// TwinCAT 3 PLC project TC3_CNCPLCBase
// Title: CNC PLC Project
// Company: Beckhoff Automation GmbH & Co. KG
// Author: Beckhoff Automation GmbH & Co. KG
// ProjectVersion: 3.1.5000.18
// Description: TwinCAT CNC Base Project
// ProgramVersion: 3.1.4022.1
// libraries:
//   Tc2_CncHli, * (Beckhoff Automation GmbH)
//   Tc2_Standard, * (Beckhoff Automation GmbH)
//   Tc2_System, * (Beckhoff Automation GmbH)
//   Tc3_CNC, * (Beckhoff Automation GmbH)
//   Tc3_EventLogger, * (Beckhoff Automation GmbH)
//   Tc3_JsonXml, * (Beckhoff Automation GmbH)
//   Tc3_Module, * (Beckhoff Automation GmbH)
// project tree:
//   CNC/ Global_CNC.TcGVL, PRG_CNCAxesHandler.TcPOU, PRG_CNCChannelHandler.TcPOU, PRG_CNCManualMode.TcPOU, PRG_CNCVariablesViewer.TcPOU, PRG_ManualFnc.TcPOU
//   / FAST.TcPOU, MAIN.TcPOU, PlcFastTask.TcTTO, PlcTask.TcTTO
//   HMI/ Global_HMI.TcGVL, ST_MachineData.TcDUT, ST_MachineMode.TcDUT, ST_MANUAL.TcDUT, ST_Position.TcDUT
//   Messages/ FB_Alarm.TcPOU, FB_ExtSimpleEventLog.TcPOU, FB_SimpleEventLog.TcPOU, Global_Messages.TcGVL, PRG_Messages.TcPOU, PRG_MessagesV2.TcPOU
//   Samples/ PRG_FastMFunctions.TcPOU
// real-time tasks:
//   TASK PlcTask: cycle T#10ms, priority 20, ADS port 350
//   TASK PlcFastTask: cycle T#10ms, priority 21, ADS port 351
// motion (NC):
//   TASK NC-Task 1 SAF: cycle T#2ms, priority 4, ADS port 501
//   TASK NC-Task 1 SVB: cycle T#10ms, priority 9, ADS port 511
//   AXIS RollerVibrator (id 1)
//     General: UnitName=Degree
//     Dynamic: AccelerationMaximum=72000, DecelerationMaximum=72000, Acceleration=72000, Deceleration=72000, Jerk=432000
//     Velo: RefSearch=313.26, RefSync=313.26, SlowManual=1566.3, FastManual=9397.8, Fast=31326, Maximum=60000
//     PositionAreaControl: Range=10
//     OtherSettings: AllowMotionCmdToSlave=true, PulseDistancePos=10, PulseDistanceNeg=10
//     encoder EncType=19
//       EncPara: ScaleFactorNumerator=360, ScaleFactorDenominator=1048576, MaxCount=#xffffffff
//     drive DrvType=16
//       DrvPara: MaxCount=#xffffffff, DriveControlDWord=#x00020000
//         Analog: VeloReferenz=36000, VeloScale=32, TorqueSetpointScale=10, ScaleFactorActTorque=0.1
//         TimeComp: TaskDelayCycles=1
//     controller CtrType=1
//       CtrPara: PriorControlFactor=1
//         PosDiffControl: Enable=false, Range=10
//         Observer: BandWidth=20
//   AXIS RollerCompactor (id 2)
//     General: UnitName=Degree
//     Dynamic: AccelerationMaximum=72000, DecelerationMaximum=72000, Acceleration=72000, Deceleration=72000, Jerk=432000
//     Velo: RefSearch=313.26, RefSync=313.26, SlowManual=1566.3, FastManual=9397.8, Fast=31326, Maximum=60000
//     PositionAreaControl: Range=10
//     OtherSettings: AllowMotionCmdToSlave=true, PulseDistancePos=10, PulseDistanceNeg=10
//     encoder EncType=19
//       EncPara: ScaleFactorNumerator=360, ScaleFactorDenominator=1048576, MaxCount=#xffffffff
//     drive DrvType=16
//       DrvPara: MaxCount=#xffffffff, DriveControlDWord=#x00020000
//         Analog: VeloReferenz=36000, VeloScale=32, TorqueSetpointScale=10, ScaleFactorActTorque=0.1
//         TimeComp: TaskDelayCycles=1
//     controller CtrType=1
//       CtrPara: PriorControlFactor=1
//         PosDiffControl: Enable=false, Range=10
//         Observer: BandWidth=20
// I/O:
//   DEVICE Device 1 (EtherCAT), AmsNetId 5.85.147.42.2.1
//     Term 1 (EK1200) [EK1200-5000 EtherCAT Power supply (2A E-Bus)]
//       Term 2 (EK1122) [EK1122 2 port EtherCAT junction]
//         Term 3 (EK1100) [EK1100 EtherCAT Coupler (2A E-Bus)]
//         Drive 4 (ctrlX DRIVE XCD (SoE) 1/2) [ctrlX DRIVE XCD (SoE) Axis 1 of 2]
//         Drive 5 (ctrlX DRIVE XCD (SoE) 2/2) [ctrlX DRIVE XCD (SoE) Axis 2 of 2]
//         Drive 6 (ctrlX DRIVE XMD (SoE) 1/2) [ctrlX DRIVE XMD (SoE) Axis 1 of 2]
//         Drive 7 (ctrlX DRIVE XMD (SoE) 2/2) [ctrlX DRIVE XMD (SoE) 2 of 2]
//         Drive 8 (ctrlX DRIVE XMD (SoE) 1/2) [ctrlX DRIVE XMD (SoE) Axis 1 of 2]
//         Drive 9 (ctrlX DRIVE XMD (SoE) 2/2) [ctrlX DRIVE XMD (SoE) 2 of 2]
//         Drive 10 (ctrlX DRIVE XMS (SoE)) [ctrlX DRIVE XMS (SoE)]
//         Drive 24 (IndraDrive MPB20 FSoE) [IndraDrive MPB20 FSoE]
//         Term 26 (EK1100) [EK1100 EtherCAT Coupler (2A E-Bus)]
//           Term 27 (EL4124) [EL4124 4Ch. Ana. Output 4-20mA, 16bit]
//           Term 28 (EL2008) [EL2008 8Ch. Dig. Output 24V, 0.5A]
//           Term 32 (EL9011) [EL9011 End Terminal]
//       Term 29 (EK1122) [EK1122 2 port EtherCAT junction]
//         Term 30 (EK1100) [EK1100 EtherCAT Coupler (2A E-Bus)]
//           Term 31 (EL7211-9014) [EL7211-9014 1Ch. MDP742 Servo motor output stage with OCT (50V, 4.5A RMS) and STO input]
//           Term 32 (EL7211-9014) [EL7211-9014 1Ch. MDP742 Servo motor output stage with OCT (50V, 4.5A RMS) and STO input]
//           Term 33 (EL9011) [EL9011 End Terminal]
//   DEVICE Device 4 (RT-Ethernet Protocol), AmsNetId 5.85.147.42.5.1
//   DEVICE Device 3 (USB)
//     Box 1 (CX2100 Power Supply)
//   DEVICE Device 5 (NOV-DP-RAM)
// variable links:
//   CNC/Axes/A <-> Device 1 (EtherCAT)/Term 1 (EK1200)/Term 2 (EK1122)/Drive 24 (IndraDrive MPB20 FSoE)
//     Inputs/Drive status word <-> AT/Drive status word
//     Inputs/Position feedback value 1 <-> AT/Position feedback value 1
//     Inputs/WcState <-> WcState/WcState
//     Outputs/Master control word <-> MDT/Master control word
//     Outputs/Position command value <-> MDT/Position command value
//   CNC/Axes/X0_M <-> Device 1 (EtherCAT)/Term 1 (EK1200)/Term 2 (EK1122)/Drive 4 (ctrlX DRIVE XCD (SoE) 1/2)
//     Inputs/Drive status word <-> AT/Drive status word
//     Inputs/Position feedback value 1 <-> AT/Position feedback value 1
//     Inputs/Power supply status word <-> AT/Power supply status word
//     Inputs/WcState <-> WcState/WcState
//     Outputs/Master control word <-> MDT/Master control word
//     Outputs/Position command value <-> MDT/Position command value
//     Outputs/Power supply control word <-> MDT/Power supply control word
//   CNC/Axes/X0_S <-> Device 1 (EtherCAT)/Term 1 (EK1200)/Term 2 (EK1122)/Drive 5 (ctrlX DRIVE XCD (SoE) 2/2)
//     Inputs/Drive status word <-> AT/Drive status word
//     Inputs/Position feedback value 1 <-> AT/Position feedback value 1
//     Inputs/WcState <-> WcState/WcState
//     Outputs/Master control word <-> MDT/Master control word
//     Outputs/Position command value <-> MDT/Position command value
//   CNC/Axes/X1_M <-> Device 1 (EtherCAT)/Term 1 (EK1200)/Term 2 (EK1122)/Drive 6 (ctrlX DRIVE XMD (SoE) 1/2)
//     Inputs/Device control: Status word <-> AT/Device control: Status word
//     Inputs/Drive status word <-> AT/Drive status word
//     Inputs/Position feedback value 1 <-> AT/Position feedback value 1
//     Inputs/WcState <-> WcState/WcState
//     Outputs/DC Bus Power Control <-> MDT/DC Bus Power Control
//     Outputs/Master control word <-> MDT/Master control word
//     Outputs/Position command value <-> MDT/Position command value
//   CNC/Axes/X1_S <-> Device 1 (EtherCAT)/Term 1 (EK1200)/Term 2 (EK1122)/Drive 7 (ctrlX DRIVE XMD (SoE) 2/2)
//     Inputs/Device control: Status word <-> AT/Device control: Status word
//     Inputs/Drive status word <-> AT/Drive status word
//     Inputs/Position feedback value 1 <-> AT/Position feedback value 1
//     Inputs/WcState <-> WcState/WcState
//     Outputs/DC Bus Power Control <-> MDT/DC Bus Power Control
//     Outputs/Master control word <-> MDT/Master control word
//     Outputs/Position command value <-> MDT/Position command value
//   CNC/Axes/Y <-> Device 1 (EtherCAT)/Term 1 (EK1200)/Term 2 (EK1122)/Drive 10 (ctrlX DRIVE XMS (SoE))
//     Inputs/Device control: Status word <-> AT/Device control: Status word
//     Inputs/Drive status word <-> AT/Drive status word
//     Inputs/Position feedback value 1 <-> AT/Position feedback value 1
//     Inputs/WcState <-> WcState/WcState
//     Outputs/DC Bus Power Control <-> MDT/DC Bus Power Control
//     Outputs/Master control word <-> MDT/Master control word
//     Outputs/Position command value <-> MDT/Position command value
//   CNC/Axes/Z_M <-> Device 1 (EtherCAT)/Term 1 (EK1200)/Term 2 (EK1122)/Drive 8 (ctrlX DRIVE XMD (SoE) 1/2)
//     Inputs/Device control: Status word <-> AT/Device control: Status word
//     Inputs/Drive status word <-> AT/Drive status word
//     Inputs/Position feedback value 1 <-> AT/Position feedback value 1
//     Inputs/WcState <-> WcState/WcState
//     Outputs/DC Bus Power Control <-> MDT/DC Bus Power Control
//     Outputs/Master control word <-> MDT/Master control word
//     Outputs/Position command value <-> MDT/Position command value
//   CNC/Axes/Z_S <-> Device 1 (EtherCAT)/Term 1 (EK1200)/Term 2 (EK1122)/Drive 9 (ctrlX DRIVE XMD (SoE) 2/2)
//     Inputs/Device control: Status word <-> AT/Device control: Status word
//     Inputs/Drive status word <-> AT/Drive status word
//     Inputs/Position feedback value 1 <-> AT/Position feedback value 1
//     Inputs/WcState <-> WcState/WcState
//     Outputs/DC Bus Power Control <-> MDT/DC Bus Power Control
//     Outputs/Master control word <-> MDT/Master control word
//     Outputs/Position command value <-> MDT/Position command value
//   NC-Task 1 SAF/Axes/RollerCompactor <-> Device 1 (EtherCAT)/Term 1 (EK1200)/Term 29 (EK1122)/Term 30 (EK1100)/Term 32 (EL7211-9014)
//     Drive/Inputs/In/nDcOutputTime <-> InfoData/DcOutputShift
//     Drive/Inputs/In/nState1 <-> DRV Statusword/Statusword
//     Drive/Inputs/In/nState2 <-> DRV Statusword/Statusword @bit 8
//     Drive/Inputs/In/nState4 @bit 1 <-> WcState/InputToggle
//     Drive/Inputs/In/nState4 <-> WcState/WcState
//     Drive/Outputs/Out/nCtrl1 <-> DRV Controlword/Controlword
//     Drive/Outputs/Out/nCtrl2 <-> DRV Controlword/Controlword @bit 8
//     Drive/Outputs/Out/nDataOut2 <-> DRV Target velocity/Target velocity
//     Enc/Inputs/In/nDataIn1 <-> FB Position/Position
//     Enc/Inputs/In/nDcInputTime <-> InfoData/DcInputShift
//     Enc/Inputs/In/nState4 @bit 1 <-> WcState/InputToggle
//     Enc/Inputs/In/nState4 <-> WcState/WcState
//   NC-Task 1 SAF/Axes/RollerVibrator <-> Device 1 (EtherCAT)/Term 1 (EK1200)/Term 29 (EK1122)/Term 30 (EK1100)/Term 31 (EL7211-9014)
//     Drive/Inputs/In/nDcOutputTime <-> InfoData/DcOutputShift
//     Drive/Inputs/In/nState1 <-> DRV Statusword/Statusword
//     Drive/Inputs/In/nState2 <-> DRV Statusword/Statusword @bit 8
//     Drive/Inputs/In/nState4 @bit 1 <-> WcState/InputToggle
//     Drive/Inputs/In/nState4 <-> WcState/WcState
//     Drive/Outputs/Out/nCtrl1 <-> DRV Controlword/Controlword
//     Drive/Outputs/Out/nCtrl2 <-> DRV Controlword/Controlword @bit 8
//     Drive/Outputs/Out/nDataOut2 <-> DRV Target velocity/Target velocity
//     Enc/Inputs/In/nDataIn1 <-> FB Position/Position
//     Enc/Inputs/In/nDcInputTime <-> InfoData/DcInputShift
//     Enc/Inputs/In/nState4 @bit 1 <-> WcState/InputToggle
//     Enc/Inputs/In/nState4 <-> WcState/WcState

CONFIGURATION TC3_CNCPLCBase
    RESOURCE PLC ON TwinCAT3
        TASK PlcFastTask(INTERVAL := T#10ms, PRIORITY := 21);
        TASK PlcTask(INTERVAL := T#10ms, PRIORITY := 20);
        PROGRAM FAST WITH PlcFastTask : FAST;
        PROGRAM MAIN WITH PlcTask : MAIN;
    END_RESOURCE
END_CONFIGURATION

// ---- HMI/ST_MachineData.TcDUT
TYPE ST_MachineData :
STRUCT
	// @1: Value1
	Value1: INT;
	// @1: Bool Value
	Value2: bool;
	// @1: Position
	pos : ST_Position;
	// @1: Manual @6:1
	manualFunction : ST_Manual;
END_STRUCT
END_TYPE

// ---- HMI/ST_MachineMode.TcDUT
TYPE ST_MachineMode :
STRUCT
	/// Operation Mode 
	Standby: BOOL;
	Manual: BOOL;
	MDI: BOOL;
	Automatic: BOOL;
	///REFERENCE		: BOOL;  TC3HR
	Homing: BOOL;
	/// Operation State
	Select : BOOL; 
	Ready  : BOOL;
	Start: BOOL;
	Stop: BOOL;
	Reset: BOOL;
	Error: BOOL;
	/// Special functions 
	ChannelSignals: ST_ChannelSignals;
	BlockSearch: ST_BlockSearch;
	SyntaxCheck: ST_SyntaxCheck;
	ManualMode: ST_ManualMode;
	/// Strings 
//	ProgramName: STRING(1024);
//	MDIString: STRING(1024);
	ProgramName: STRING(HLI_IMCM_MODE_STATE_PARAM_STRL);
	MDIString: STRING(HLI_IMCM_MODE_STATE_PARAM_STRL);

END_STRUCT
END_TYPE

// ---- HMI/ST_MANUAL.TcDUT
TYPE ST_MANUAL :
STRUCT
	// @1:cylinder one @2:on:1 @3:off:1 @4:pos1:1 @5:pos2:0
	cyl1 			: BYTE;	
	cyl1Status		: BYTE;
	
	// @1:conveyor @2:IMG1:1 @2:IMG2 @3:IMG15 @4:IMG16 @5:IMG7 @6:IMG13 @7:IMG14
	conv 			: BYTE;
	convStatus 		: BYTE;
	
	
END_STRUCT
END_TYPE

// ---- HMI/ST_Position.TcDUT
TYPE ST_Position :
STRUCT
	// @1:X
	x	:	LREAL;
	// @1:Y
	y	: 	LREAL;
	// @1:Z	
	Z	: 	LREAL;
END_STRUCT
END_TYPE

// ---- CNC/Global_CNC.TcGVL
VAR_GLOBAL CONSTANT
	// Max index of channel that is used starting at 0, example: 1 -> totally 2 channels, maximum of 11 (12 channels) is allowed here
	MAX_USED_CHANNEL_IDX		: INT := 2;									
	libVersion					: ST_LibVersion := stLibVersion_Tc3_CNC;  	 
END_VAR

// ---- HMI/Global_HMI.TcGVL
VAR_GLOBAL
	/// HMI -> PLC 
	PLCChannelSignals: ST_ChannelSignals;
	/// HMI -> PLC 
	PLCSelectedChannel: INT := 0;
	/// HMI -> PLC 
	PLCFeedOverride: UINT := 100;
	/// HMI -> PLC 
	PLCSpindleOverride: UINT := 100;
	/// HMI -> PLC 
	PLCAxisEnable: BOOL;
	/// PLC -> HMI  
	PLCStatusAxisEnabled : BOOL;	
	/// HMI -> PLC 
	PLCReset: BOOL;
	PLCMachineMode: ARRAY[0..MAX_USED_CHANNEL_IDX] OF ST_MachineMode;
	/// PLC -> HMI : angewähltes File 
	PLCToHmiFile: STRING(255);
	/// Variablen für das Module "InformPlc" 
	bToggle: BOOL;
	sActualForm: STRING(255);
	nUserLevel: INT;
	sUserName: STRING(255);
	/// steigende Flanke: Applikation beenden 
	bExitApp: BOOL;	
	
	userActivity : BOOL;
	
	// @1:MachineData
	MachineData : ST_MachineData;
	
	// spindle manual mode
	nSpindleRpm:	DINT;	
	bSpindleStart: BOOL;
	bSpindleStop: BOOL;
	
	ManualFnc : ARRAY[0..3] OF FB_ManualFncFull;
	
END_VAR

// ---- Messages/Global_Messages.TcGVL
VAR_GLOBAL
	///--------------------------
	///	Messages                
	///--------------------------
	MSG_WARNING_List: ARRAY[FIRST_MESSAGE..LAST_MESSAGE] OF BOOL;
	MSG_WARNING_ListQuit: ARRAY[FIRST_MESSAGE..LAST_MESSAGE] OF BOOL;	
	MSG_ALARM_List: ARRAY[FIRST_MESSAGE..LAST_MESSAGE] OF BOOL;
	MSG_ALARM_ListQuit: ARRAY[FIRST_MESSAGE..LAST_MESSAGE] OF BOOL;			
END_VAR

VAR_GLOBAL CONSTANT
	FIRST_MESSAGE: UDINT := 1;
	LAST_MESSAGE: UDINT := 50;	
END_VAR

// ---- FAST.TcPOU
PROGRAM FAST
VAR
	nChan : INT;
	MOS_TS: INT;
	i: INT;	
	ChannelMHTFunction : ARRAY[0..MAX_USED_CHANNEL_IDX] OF HLI3_QuitChannelMHTFunction;
END_VAR

(****************************************************************************************)
(*	  							Wait for HLI initialization								*)
(****************************************************************************************)
IF NOT CNCSystem.bHLIInit THEN
	RETURN;
END_IF

IF PRG_CNCChannelHandler.stOptions.bDisableMFunctHandling THEN
	FOR i := 0 TO MAX_USED_CHANNEL_IDX DO
		ChannelMHTFunction[i](nChanIdx:=0, bM30Acknowledgement := TRUE);
	END_FOR
END_IF	

(* Programm call for MOS_TS M functions *)
// PRG_FastMFunctions();

END_PROGRAM

// ---- CNC/PRG_CNCChannelHandler.TcPOU
PROGRAM PRG_CNCChannelHandler
VAR	
	nChan					: INT;
	nOldSelectedChannel		: UDINT;
	CNCChannel				: ARRAY[0..MAX_USED_CHANNEL_IDX] OF HLI3_CNCChannel;	
	BlockSearch_Channel		: ARRAY[0..MAX_USED_CHANNEL_IDX] OF HLI3_BlockSearch;
	ErrorHandler_Channel	: ARRAY[0..MAX_USED_CHANNEL_IDX] OF FB_ChannelError;
	nChanNo: UDINT;	
	i: INT;	
	stOptions				: ST_CNC_CH_Options;
END_VAR

(****************************************************************************************)
(* POU:		PRG_ChannelHandler                     										*)
(* Type:	PRG																			*)
(* Author: 	HR / TV / MiB                                          						*)
(* Date: 	23.01.11																	*)
(* Last:	29.03.18																	*)
(* Rev.: 	1.6                                              							*)
(* ------------------------------------------------------------------------------------ *)
(* Desc:	Description																	*)
(****************************************************************************************)

(****************************************************************************************)
(*	  Map CNC function selection from HMI to selected channel (and state vice versa)  	*)
(****************************************************************************************)
IF (nOldSelectedChannel <>INT_TO_UDINT(PLCSelectedChannel)) THEN
	PLCChannelSignals.SingleBlock 		:= PLCMachineMode[PLCSelectedChannel].ChannelSignals.SingleBlock;
	PLCChannelSignals.PrgBlockIgnore	:= PLCMachineMode[PLCSelectedChannel].ChannelSignals.PrgBlockIgnore;
	PLCChannelSignals.M01Stop 			:= PLCMachineMode[PLCSelectedChannel].ChannelSignals.M01Stop;
	PLCChannelSignals.Backward 			:= PLCMachineMode[PLCSelectedChannel].ChannelSignals.Backward;
	PLCChannelSignals.FeedHold 			:= PLCMachineMode[PLCSelectedChannel].ChannelSignals.FeedHold;
	nOldSelectedChannel 				:= INT_TO_UDINT(PLCSelectedChannel);
END_IF

PLCMachineMode[PLCSelectedChannel].ChannelSignals.SingleBlock 		:= PLCChannelSignals.SingleBlock;
PLCMachineMode[PLCSelectedChannel].ChannelSignals.PrgBlockIgnore 	:= PLCChannelSignals.PrgBlockIgnore;
PLCMachineMode[PLCSelectedChannel].ChannelSignals.M01Stop 			:= PLCChannelSignals.M01Stop;
PLCMachineMode[PLCSelectedChannel].ChannelSignals.Backward 		:= PLCChannelSignals.Backward;
PLCMachineMode[PLCSelectedChannel].ChannelSignals.FeedHold 		:= PLCChannelSignals.FeedHold;


stOptions.bReferenceModeStartRequired := FALSE;

FOR i := 0 TO MAX_USED_CHANNEL_IDX DO
		
	nChan := i;	
	IF (HLI3_CheckChannelValid(nChan)) THEN		
		
		(* Error handler for channel 1 *)
		ErrorHandler_Channel[nChan](nChanIdx			:= nCHan);				
				
		(* Channel interface *)
		CNCChannel[nChan]
			(nChanIdx			:= nChan,							
			 // Operation Mode with VAR_IN_OUT Variables 
			 bModeStandby		:= PLCMachineMode[nChan].Standby,
			 bModeAutomatic		:= PLCMachineMode[nChan].Automatic,
			 bModeManual		:= PLCMachineMode[nChan].Manual,
			 bModeMDI			:= PLCMachineMode[nChan].MDI,	 
			 bModeReference		:= PLCMachineMode[nChan].Homing,
			 // Operation State with VAR_IN_OUT Variables
			 bStateSelect		:= PLCMachineMode[nChan].Select,
			 bStateReady		:= PLCMachineMode[nChan].Ready,
			 bStateStart		:= PLCMachineMode[nChan].Start,
			 bStateStop			:= PLCMachineMode[nChan].Stop,
			 bStateReset		:= PLCMachineMode[nChan].Reset,
			 // Operation Mode with VAR_IN Varaibles, the command is executed with a rising edge 
			 bCmdAutomatic 		:= FALSE,
			 bCmdManual 		:= FALSE,
    		 bCmdReference 		:= FALSE,
    		 bCmdMDI 			:= FALSE,		
			 // Operation State with VAR_IN Varaibles, the command is executed with a rising edge
			 bCmdStart 			:= FALSE,
			 bCmdStop  			:= FALSE,
	         bCmdReset 			:= FALSE,					 			 
			 // EmergencyStop 
			 bEmergencyStop 	:= FALSE,		(* If TRUE the interpolation will be aborted, Signal is no TwinSAFE function !*)
			 // Override 
			 nFeedOverride		:= PLCFeedOverride * 10,
			 nRapidFeedOverride := PLCFeedOverride * 10, 
			 // Special Functions 
			 sProgramName		:= PLCMachineMode[nChan].ProgramName,			 
			 sMDIString			:= PLCMachineMode[nChan].MDIString,
			 bBackwardMotion	:= PLCMachineMode[nChan].ChannelSignals.Backward,
			 bPrgBlockIgnore	:= PLCMachineMode[nChan].ChannelSignals.PrgBlockIgnore,
			 bFeedHold			:= PLCMachineMode[nChan].ChannelSignals.FeedHold,
			 bSingleBlock		:= PLCMachineMode[nChan].ChannelSignals.SingleBlock,
			 bDoSingleBlock		:= PLCMachineMode[nChan].ChannelSignals.DoSingleBlock,
			 bM01Stop			:= PLCMachineMode[nChan].ChannelSignals.M01Stop,
			 nSyntaxCheck		:= PLCMachineMode[nChan].SyntaxCheck.nType,
			 bM30Acknowledgement:= TRUE,
			 // Manual Mode 			 						 
			 stManualModeParameter  	 	 := stManualModeParameter[nChan],
			 stManualModeControlElements	 := stManualModeControlElements[nChan],
			 stManualModeControlElementState := stManualModeControlElementState,
			 // Options
			 stOptions			:= 	stOptions			 			 
			);
		
		(* Handle block search *)
		BlockSearch_Channel[nChan]
			(nChanIdx			:= nChan,
			 bStartRead      	:= PLCMachineMode[nChan].BlockSearch.bStartRead,   (* Edge signal *)
			 bStartWrite     	:= PLCMachineMode[nChan].BlockSearch.bStartWrite,  (* Edge signal *)
			 BlockSearch		:= PLCMachineMode[nChan].BlockSearch
			);
		
		CNCSystem.Channel[nChan].ActDistance 	:= DINT_TO_LREAL(BlockSearch_Channel[nChan].coveredDistance_AfterReset) / 10.0;
		CNCSystem.Channel[nChan].ActBlockCount 	:= BlockSearch_Channel[nChan].actualBlockCount_AfterReset;
						
	END_IF
END_FOR

END_PROGRAM

// ---- MAIN.TcPOU
PROGRAM MAIN
VAR
  
END_VAR

HLI3_Init(); 
PRG_Messages();  	// Messages Eventlogger V1
PRG_MessagesV2();   // Messages Eventlogger V2

(* Call CNC related code only if the HLI has been initialized succesfully! *)
IF CNCSystem.bHLIInit THEN
	PRG_CNCAxesHandler();    	
	PRG_CNCManualMode();
	PRG_CNCChannelHandler();	
	PRG_CNCVariablesViewer();
	PRG_ManualFnc();		
END_IF
(* Reset the reset flag from HMI *)
PLCReset := FALSE;

END_PROGRAM

// ---- Messages/PRG_Messages.TcPOU
PROGRAM PRG_Messages
VAR
	bStart: BOOL;
	fbWarningMessages : FB_SimpleEventLog;
	fbAlarmMessages : FB_SimpleEventLog;
	//fbExAlarmMessages : FB_ExtSimpleEventLog;
END_VAR

(*
	TCEVENTCLASS_NONE			:=0,	 No class
	TCEVENTCLASS_MAINTENANCE	:=1,	 Maintenance hint
	TCEVENTCLASS_MESSAGE		:=2,	 Message
	TCEVENTCLASS_HINT			:=3,	 Hint
	TCEVENTCLASS_STATEINFO		:=4,	 State information
	TCEVENTCLASS_INSTRUCTION	:=5,	 Instruction
	TCEVENTCLASS_WARNING		:=6,	 Warning
	TCEVENTCLASS_ALARM			:=7,	 Alarm
	TCEVENTCLASS_PARAMERROR		:=8	 Parameter error
*)


(* Shows how to generate messages *)
IF NOT bStart THEN
	bStart 				:= TRUE;

	fbWarningMessages
		(Init			:= TRUE,
		 SourceId		:= 51,
		 Class			:= TCEVENTCLASS_WARNING,
		 QuitRequireD	:= FALSE,
		 adrAlarmArray	:= ADR(MSG_WARNING_List),
		 adrQuitArray	:= ADR(MSG_WARNING_ListQuit)
		);

	fbAlarmMessages
		(Init			:= TRUE,
		 SourceId		:= 50,
		 Class			:= TCEVENTCLASS_ALARM,
		 QuitRequired	:= FALSE,
		 adrAlarmArray 	:= ADR(MSG_ALARM_List),
		 adrQuitArray	:= ADR(MSG_ALARM_ListQuit)
		);
		(*
		fbExAlarmMessages(
			Init:= TRUE, 
			SourceId:= 52,
			Class:= TCEVENTCLASS_WARNING, 				
			QuitRequired:= FALSE, 
			adrAlarmArray:= ADR(MSG_ExALARM_List), 
			adrQuitArray:= ADR(MSG_ExALARM_ListQuit), 
			adrEventData:= ADR(MSG_ExALARM_EventData),	 
			sFormatString:= '%d%s'		  
			);
			*)
ELSE
	fbWarningMessages
		(Init			:= FALSE);

	fbAlarmMessages
		(Init			:= FALSE);	
		(*
	fbExAlarmMessages
		(Init			:= FALSE);
*)	
END_IF

END_PROGRAM

// ---- Messages/FB_SimpleEventLog.TcPOU
///****************************************************************************************
///Name:				FB_SimpleEventLog
///Date:				13.10.2004
///Author:			Dirk Nordberg (BECKHOFF INDUSTRIE ELEKTRONIK)
///
///Description: Function block to control the EventLogger
///	Messages can be activated or deactivated through an array of bool.
///	The subscription of the array is equivalent to EventID from EventLogger.
///	Function block will be initialized with Init flag, then the busy flag is set true. 
///
///	Revision:	1.4
///	History:		13.10.2004	Ng	start coding
///					17.04.2005	MK	runtime optimized
///					07.07.2005	MK	short puls BF
///				    29.11.2010 	MiB  quittierungspflichtige Merker funktionieren nun wieder
///                 21.06.2013  TV   change : data type for pointer address from uint to pointer of int 
///****************************************************************************************
FUNCTION_BLOCK FB_SimpleEventLog
VAR_INPUT
	/// Rising flag starts the initialization 
	Init: BOOL;
	/// Number of the source Id 
	SourceId: UINT;
	/// Alarm error class 
	Class: UINT;
	/// Activate or deaktivate confirmation 
	QuitRequired: BOOL;
	/// Adress of the array for the messages 
	adrAlarmArray: POINTER TO BOOL;
	/// ...with constant boundaries ARRAY_LBOUND to ARRAY_UBOUND for array size 
	adrQuitArray: POINTER TO BOOL;
END_VAR
VAR_OUTPUT
	Busy: BOOL;
	Err: BOOL;
	ErrId: UDINT;
END_VAR
VAR CONSTANT
	ARRAY_LBOUND: UDINT := FIRST_MESSAGE;
	ARRAY_UBOUND: UDINT := LAST_MESSAGE;
	TCEVENTDATAFORMATSTRING: STRING := ' ';
	STATE_INIT: INT := 0;
	STATE_IDLE: INT := 1;
	STATE_RESET_EVENT: INT := 2;
	STATE_QUIT_EVENT: INT := 3;
	STATE_RESET_END: INT := 4;
	STATE_WAIT: INT := 5;
END_VAR
VAR
	state: INT;
	///{flag nowatch on }
	bReady: BOOL := TRUE;
	nMsgHasChanged: DINT;
	bEvtState: ARRAY[ARRAY_LBOUND..ARRAY_UBOUND] OF BOOL;
	event: ARRAY[ARRAY_LBOUND..ARRAY_UBOUND] OF ADSLOGEVENT;
	idx: UDINT;
	CfgEvent: TcEvent;
	bWait: BOOL;
	ptAlarm: POINTER TO BOOL;
	ptQuit: POINTER TO BOOL;
	RT_Init: R_TRIG;
END_VAR

nMsgHasChanged := MEMCMP(ADR(bEvtState), adrAlarmArray, SIZEOF(bEvtState));

RT_Init(CLK:=Init);

CASE State OF
	STATE_INIT:		(* Set the parameter for TcEvent *)
		Err := FALSE;
		ErrId :=0;
		Busy := FALSE;
		CfgEvent.Prio := 0;
		CfgEvent.DataFormatStrAddress := ADR(TCEVENTDATAFORMATSTRING);
		// CfgEvent.Flags := TCEVENTFLAG_LOG OR TCEVENTFLAG_SRCID OR TCEVENTFLAG_PRIOCLASS OR TCEVENTFLAG_FMTSELF OR 16#1000;
		// MiB 2015.10.07 Flags changed -> now the class is defined here and not in Event config file.
		CfgEvent.Flags := TCEVENTFLAG_LOG OR TCEVENTFLAG_SRCID;
		CfgEvent.StreamType := TCEVENTSTREAM_SIMPLE;
		CfgEvent.ProgId := 'TcEventFormatter.TcXmlFormatter';
		CfgEvent.SourceId := SourceId;
		CfgEvent.Class := Class ;
		CfgEvent.bQuitRequired := QuitRequired;
		FOR idx := ARRAY_LBOUND TO ARRAY_UBOUND BY 1 DO
			CfgEvent.Id := idx;
			event[idx](NETID:='', PORT:=110, Event:=FALSE , EventQuit:=FALSE,
				 EventConfigData:=CfgEvent, FbCleanup:=FALSE, TMOUT:=t#1s);
		END_FOR;
		State := STATE_IDLE;

	STATE_IDLE:
		(* nothing to do *)
		IF nMsgHasChanged = 0
			AND  NOT QuitRequired
			AND bReady = TRUE
			AND NOT RT_Init.Q THEN
			RETURN;
		END_IF

		IF adrAlarmArray <> 0 THEN
			ptAlarm := adrAlarmArray;
			IF CfgEvent.bQuitRequired AND adrQuitArray <> 0 THEN
				ptQuit := adrQuitArray;
				FOR idx := ARRAY_LBOUND TO ARRAY_UBOUND BY 1 DO
					event[idx](Event:=ptAlarm^, EventQuit:=ptQuit^);
					ptAlarm := ptAlarm + 1;
					ptQuit := ptQuit + 1;
				END_FOR;
				bReady := TRUE;
			ELSE
				bReady := TRUE;
				FOR idx := ARRAY_LBOUND TO ARRAY_UBOUND BY 1 DO
					event[idx](Event:=ptAlarm^);
					IF (NOT (ptAlarm^ = TRUE
							AND event[idx].Event = TRUE		(* event is set/on *)
							AND event[idx].Quit = FALSE
							AND event[idx].EventState = TCEVENTSTATE_SIGNALED)
						AND NOT (ptAlarm^ = FALSE
							AND event[idx].Event = FALSE		(* event is reset/off *)
							AND event[idx].Quit = TRUE
							AND event[idx].EventState = TCEVENTSTATE_INVALID)) THEN
						bReady := FALSE;
					END_IF
					ptAlarm := ptAlarm + 1;
				END_FOR;

				(* copy the status *)
				IF bReady THEN
					MEMCPY(ADR(bEvtState), adrAlarmArray, SIZEOF(bEvtState));
				END_IF

			END_IF
		END_IF

		IF RT_Init.Q THEN
			Busy := TRUE;
			State := STATE_RESET_EVENT;
		END_IF

	STATE_RESET_EVENT:(*---------------------------------- clear messages ----------------------------------------*)
		FOR idx := ARRAY_LBOUND TO ARRAY_UBOUND BY 1 DO
			IF event[idx].EventState = TCEVENTSTATE_SIGNALED THEN
				event[idx](Event:=FALSE, EventQuit:= FALSE, FbCleanup:= FALSE, TMOUT:= t#1s);
				IF event[idx].Err THEN
					Err := TRUE;
					ErrId := event[idx].ErrId;
					IF event[idx].ErrId = 1282 THEN	(* Message Router: mailbox full *)
						event[idx](Event:=FALSE, EventQuit:= FALSE, FbCleanup:= FALSE);
						RETURN;
					END_IF
				END_IF
			END_IF;
		END_FOR;
		State := STATE_QUIT_EVENT;

	STATE_QUIT_EVENT:(*---------------------------------- quit messages ----------------------------------------*)
		FOR idx := ARRAY_LBOUND TO ARRAY_UBOUND BY 1 DO
			IF event[idx].EventState = TCEVENTSTATE_SIGNALED THEN
				event[idx](Event:=FALSE, EventQuit:= TRUE, FbCleanup:= FALSE, TMOUT:= t#1s);
				IF event[idx].Err THEN
					Err := TRUE;
					ErrId := event[idx].ErrId;
					IF event[idx].ErrId = 1282 THEN	(* Message Router: mailbox full *)
						event[idx](Event:=FALSE, EventQuit:= FALSE, FbCleanup:= FALSE);
						RETURN;
					END_IF
				END_IF
			END_IF;
		END_FOR;
		State := STATE_RESET_END;

	STATE_RESET_END:
		bWait := FALSE;
		FOR idx := ARRAY_LBOUND TO ARRAY_UBOUND BY 1 DO
			event[idx](Event:=FALSE, EventQuit:= FALSE, FbCleanup:= FALSE);
			IF event[idx].EventState = TCEVENTSTATE_SIGNALED THEN
				bWait := TRUE;
			END_IF
		END_FOR;
		IF NOT bWait THEN
			State := STATE_INIT;
		END_IF

END_CASE

END_FUNCTION_BLOCK

// ---- Messages/PRG_MessagesV2.TcPOU
PROGRAM PRG_MessagesV2
VAR
	arrAlarmSimple: ARRAY[1..10] OF FB_Alarm;	
	bTestAlarm1: BOOL;
	bTestAlarm2: BOOL;
	bTestAlarm3: BOOL;
	sTestString : STRING := 'this is a test line';
END_VAR

;

(* add Alarms.tmc to "Systen\Type System" before uncommenting this *)

(*
arrAlarmSimple[1](Event := TC_EVENTS.Alarms.Alarm1);
arrAlarmSimple[1].Raise := bTestAlarm1;
arrAlarmSimple[1].AddInfo := sTestString;


arrAlarmSimple[2](Event := TC_EVENTS.Alarms.Alarm2);
arrAlarmSimple[2].Raise := bTestAlarm2;

arrAlarmSimple[3](Event := TC_EVENTS.Alarms.Alarm3);
arrAlarmSimple[3].Raise := bTestAlarm3;
*)

END_PROGRAM

// ---- Messages/FB_Alarm.TcPOU
FUNCTION_BLOCK FB_Alarm
VAR_INPUT
	Event : TcEventEntry;  // AlarmEntry from TMS Editor. Example: TC_EVENTS.Alarms.Alarm1
	Raise : BOOL;		   // true -> Alarm is active, false -> Alarm not active
	AddInfo: STRING;	   // if <> empty -> additional Info that is transfered together with alarm
END_VAR
VAR_OUTPUT
END_VAR
VAR
	_alarm : FB_TcAlarm;
	_initDone : BOOL;
	_rTrigRaise : R_TRIG;
	_fTrigRaise : F_TRIG;
	_fbSourceInfo : FB_TcSourceInfo;
	_fbJson      : FB_JsonSaxWriter;
	_sJsonDoc    : STRING(255);	
END_VAR

(* ========================================================= *)
(*    FUN: FB_Alarm                   					     *)
(* --------------------------------------------------------- *)
(*   Desc: Simple usage of Eventlogger2 Alarms               *)
(* Author: MiB                                               *)
(*   Date: 09.03.2021                                        *)
(*   Rev.: 1.0                                               *)
(* ========================================================= *)


// init
IF NOT _initDone AND Event.nEventId <> 0 THEN
	_fbSourceInfo.sName := 'PLC';
	_alarm.CreateEx(Event, FALSE, _fbSourceInfo );
	_initDone := TRUE;
END_IF

// raise alarm
_rTrigRaise(clk := Raise);
IF _rTrigRaise.Q AND NOT _alarm.bRaised  THEN
	IF LEN(AddInfo) > 0 THEN 
		_fbJson.ResetDocument();
		_fbJson.StartObject();
		_fbJson.AddKey('AddInfo');
		_fbJson.AddString(AddInfo);		
		_fbJson.EndObject();
		_sJsonDoc := _fbJson.GetDocument();
	    _alarm.SetJsonAttribute(_sJsonDoc);		
	ELSE
		_alarm.SetJsonAttribute('');
	END_IF
	_alarm.Raise(0);
END_IF

// clear alarm
_fTrigRaise(clk := Raise);
IF _fTrigRaise.Q AND _alarm.bRaised THEN
	_alarm.Clear(0, FALSE);
END_IF

END_FUNCTION_BLOCK

// ---- CNC/PRG_CNCAxesHandler.TcPOU
PROGRAM PRG_CNCAxesHandler
VAR
	nHliAxisIdx					: INT;				
	fbCNC_Axis					: ARRAY[0..HLI_SYS_AX_MAXIDX] OF FB_CNCAxis;	
	
	nFirstSpindle				: INT := -1;
	fbHandleSpindleTechno		: HLI3_HandleSpindleTechnoGearChange;
	M3,M4,M5,M19				: BOOL;
	MDummy						: BOOL;
	M40, M41, M42, M43, M44, M45: BOOL;
	
	fbAxesError 				: FB_AxesError;
		
	// FB_CNCAxis Sample
	// fbAxis_X 					:  FB_CNCAxis; 
	// stParameter					:  ST_CNC_AX_Parameter;
	// stOptions					:  ST_CNC_AX_Options;
	// stPLCopen					:  ST_CNC_AX_PLCopen;
			
	(*
	fbHandleSpindleTechnoPlcSp	: HLI3_HandleSpindleTechno;
	SM3,SM4,SM5,SM19			: bool; 
	*)
	bCalibrationCam: BOOL;
	fbMoveSpindle: HLI3_MoveSpindle;
END_VAR

(****************************************************************************************)
(* POU:		PRG_AxesHandler                     										*)
(* Type:	PRG																			*)
(* Author: 	TV,MiB                                             							*)
(* Date: 	20.02.2019																	*)
(* Rev.: 	1.6                                               							*)
(* ------------------------------------------------------------------------------------ *)
(* Desc:	Description																	*)
(****************************************************************************************)

fbAxesError(bReset := PLCReset);

(****************************************************************************************)
(*							Release of all reachable axes								*)
(****************************************************************************************)
PLCStatusAxisEnabled := TRUE;   
FOR nHliAxisIdx := 0 TO UDINT_TO_INT(gNrAx-1) DO			
	fbCNC_Axis[nHliAxisIdx](
		nLogAxisNo :=  UINT_TO_INT(gpAx[nHliAxisIdx]^.head.log_ax_nr_r),
		bEnable		:= PLCAxisEnable);
		IF (NOT fbCNC_Axis[nHliAxisIdx].stStatus.bIsEnabled) THEN    // if one axis status is "not enabled" -> reset PLCStatusAxisEnabled
			PLCStatusAxisEnabled := FALSE;
		END_IF
		IF HLI3_CheckAxisValid(nHliAxisIdx) THEN
			IF nFirstSpindle = -1 AND gpAx[nHliAxisIdx]^.ipo_state.spindle_axis_r THEN  (* store HLIIndex of first spindle *)
				nFirstSpindle := nHliAxisIdx;
			END_IF
		END_IF
END_FOR


	// FB_CNCAxis Sample 

	// CNC Axis Options
	
	// stOptions.strPathCompTable;
	// stOptions.bActivateCompTable;
	// stOptions.bProbingSignal;
	// stOptions.bReducedSpeed;
	// stOptions.bReducedSpeedZone1;
	// stOptions.bReducedSpeedZone2;
	// stOptions.bResetCalibration;
	
	// CNC Parameters
			
	// stParameter.bWriteParameter;
	// stParameter.nNumParameters  	:= 2;
	// stParameter.strTempPath		:= 'C:\';
	
	// stParameter.ParamList[0].strName 	:= 'kenngr.swe_pos';
	// stParameter.ParamList[0].strValue 	:= '30000000';

	// stParameter.ParamList[1].strName 	:= 'kenngr.swe_neg';
	// stParameter.ParamList[1].strValue 	:= '0';

	// PLCOpen
	// stPLCopen.nOverride;
	// stPLCopen.bExecuteHoming;
	// stPLCopen.bCamSignal;
	// stPLCopen.bExecuteMoveAbsolute;
	// stPLCopen.bExecuteReset;
	// stPLCopen.fPosition;
	// stPLCopen.fVelocity;
	// stPLCopen.fAcceleration;
	// stPLCopen.fJerk;
	
	(*
	fbAxis_X(
		nLogAxisNo:=1, 
		bEnable:= PLCAxisEnable, 
		bCalibrationCam:= bCalibrationCam, 
		bSetRefOffset:= , 
		fRefOffset:= , 
		bFeedhold:= ,
		stOptions:= stOptions, 
		stParameter:= stParameter, 
		stPLCopen:= stPLCopen, 
		stStatus=> );
*)		
 

(* if there exits spindles use the first one for spindleoverride *)
IF nFirstSpindle <> -1 THEN
	HLI3_SetAxisOverride(nHliAxisIdx:= nFirstSpindle , nOverride:= PLCSpindleOverride *10);

	fbHandleSpindleTechno(
		nHliAxisIdx:=nFirstSpindle , 		
		bIsChannelSpecific:= FALSE, 
		bHandleGearChange := FALSE,		
		nRevolution=> , 
		nPosition=> , 
		bError=> , 
		nErrorId=> , 
		M03:= M3, 
		M04:= M4, 
		M05:= M5, 
		M19:= M19,
		M40 := M40,
		M41 := M41,
		M42 := M42,
		M43 := M43,
		M44 := M44,
		M45 := M45,
		); 
	(* acknowledge all spindle M funnctions immediately *)
	M3 := FALSE;  
	M4 := FALSE;
	M5 := FALSE;
	M19 := FALSE;
	
	
	
	(* Example for starting and stopping a spindle in manual mode in first channel *)
	IF (CNCSystem.Channel[0].ActMode = HLI_IMCM_MANUAL_MODE) THEN 	
		fbMoveSpindle(
			nHliAxisIdx:=nFirstSpindle , 
			nSpeed:= nSpindleRpm ,   (* defined in Global_HMI *)
			bStart:=bSpindleStart, 	 (* defined in Global_HMI *)
			bStop:= bSpindleStop , 	 (* defined in Global_HMI *)
			bBusy=> , 
			bError=> , 
			nErrID=> , 
			sErrText=> );
	END_IF
	IF (bSpindleStart AND NOT fbMoveSpindle.bBusy) THEN 
		bSpindleStart := FALSE;
	END_IF
	IF (bSpindleStop AND NOT fbMoveSpindle.bBusy) THEN 
		bSpindleStop := FALSE;
	END_IF	
	
	
END_IF



(* Howto use plc controlled spindle : *)
(*
fbHandleSpindleTechnoPlcSp(
	nHliAxisIdx:= 0 , 
	nHliChannelIdx:= 0 , 
	bIsChannelSpecific:= TRUE, 
	nLogAxisNoChannelSpecific:= 95 , 
	bHandleGearChange:= FALSE , 
	bChannelReset:= FALSE, 
	nRevolution=> , 
	nPosition=> , 
	bError=> , 
	nErrorId=> , 
	M03:= SM3, 
	M04:= SM4, 
	M05:= SM5, 
	M19:= SM19);
*)

END_PROGRAM

// ---- CNC/PRG_CNCManualMode.TcPOU
PROGRAM PRG_CNCManualMode
VAR
	fbUintUdInt: ARRAY [0..MAX_USED_CHANNEL_IDX] OF FB_Uint_Udint;
	nHandwheel : UINT;		(* increments for handwheel (e.g. EL5101   *)
	nHandWheelBig: UDINT;
	i: INT;
END_VAR


FOR i := 0 TO MAX_USED_CHANNEL_IDX DO
	
	IF (HLI3_CheckChannelValid(i)) THEN

		stManualModeParameter[i].stChannelParameter.nChanIdx						:= i;       (* Channel 1 *)
		stManualModeParameter[i].stChannelParameter.nInc							:= PLCMachineMode[i].ManualMode.nInc * 10;
		stManualModeParameter[i].stChannelParameter.bG200ConfigurationViaPLC		:= TRUE;		
		
		stManualModeParameter[i].stChannelParameter.eManualType						:= UINT_TO_INT(PLCMachineMode[i].ManualMode.nManualTyp);			
		IF (stManualModeParameter[i].stChannelParameter.eManualType = E_CNC_ManualType.Handwheel AND i <> PLCSelectedChannel) THEN	(* if in Handwheel mode and the channel is NOT selected -> leave handwheel mode and change to TippMode*)
			stManualModeParameter[i].stChannelParameter.eManualType						:= E_CNC_ManualType.TippMode;
		END_IF		
		
		stManualModeParameter[i].stChannelParameter.stManualOption.bTrafoActive := PLCMachineMode[i].ManualMode.stManualOption.bTrafoActive;
        stManualModeParameter[i].stChannelParameter.stManualOption.bEcsActive := PLCMachineMode[i].ManualMode.stManualOption.bEcsActive;
        stManualModeParameter[i].stChannelParameter.stManualOption.eZeroOffset := PLCMachineMode[i].ManualMode.stManualOption.eZeroOffset;
							
		
		stManualModeParameter[i].stChannelParameter.nHandwheelResolution			:= UDINT_TO_DINT(PLCMachineMode[i].ManualMode.nHwResolution);    (* 0.1 µm /rev (from HMI) *)						
		stManualModeParameter[i].stAxisParameter.stControlUnit[0].nLogAxisNr		:= PLCMachineMode[i].ManualMode.nLogAxisNumber;   (* Log. Achs Nummer *)
		IF stManualModeParameter[i].stAxisParameter.stControlUnit[0].nLogAxisNr = 0 THEN
			stManualModeParameter[i].stAxisParameter.stControlUnit[0].nLogAxisNr := gpCh[i]^.bahn_state.coord_r[0].log_achs_nr_r;
			PLCMachineMode[i].ManualMode.nLogAxisNumber := gpCh[i]^.bahn_state.coord_r[0].log_achs_nr_r;
		END_IF
		stManualModeParameter[i].stAxisParameter.stControlUnit[0].nSpeed			:= LREAL_TO_UDINT(PLCMachineMode[i].ManualMode.nSpeed * 16.666);
		stManualModeControlElements[i].stControlKeys[0].bKeyNeg						:= PLCMachineMode[i].ManualMode.bKeyNeg;
		stManualModeControlElements[i].stControlKeys[0].bKeyPos						:= PLCMachineMode[i].ManualMode.bKeyPos;
		stManualModeControlElements[i].stControlKeys[0].bKeyRapid					:= PLCMachineMode[i].ManualMode.bKeyRapid;
		
		(* the cnc needs an UDINT for handwheel increments, fbUintUdint extends an UInt to an UDINT *)
		(* the resoltion of the handwheel is parameterized in CNC-Task GEO/Manual MDS: (e.g. 400 handwheel inc / handwheel revolution
		
				hr_data[0].hr_aufl_z              400         ( P-MANU-00005 : Handwheel resolution numerator
				hr_data[0].hr_aufl_n                1     	  ( P-MANU-00006 : Handwheel resolution denominator
		*) 
		fbUintUdInt[i](nInSmall := nHandwheel, nBig := nHandWheelBig);
		stManualModeControlElements[i].nHandwheelInc[0] :=  UDINT_TO_DINT(nHandWheelBig);
  END_IF
END_FOR

END_PROGRAM

// ---- CNC/PRG_CNCVariablesViewer.TcPOU
PROGRAM PRG_CNCVariablesViewer
VAR			
	fbReadCNCVariables : FB_ReadCNCVariables;		
END_VAR

fbReadCNCVariables(
	bEnable:= TRUE, 
	nChanIdx:= PLCSelectedChannel, 
	eVariablesType:= eVariablesType, 
	tIntervall:= T#1S, 	 
	stCNCVariablesViewer_Data:= stCNCVariablesViewer_Data);

END_PROGRAM

// ---- CNC/PRG_ManualFnc.TcPOU
PROGRAM PRG_ManualFnc
VAR
END_VAR



	ManualFnc[0].headerText := 'HeaderText 1';
	ManualFnc[0].addText := 'addText';
	ManualFnc[0].infoText1 := 'infoText1';
	ManualFnc[0].infoText2 := 'infoText2';
	ManualFnc[0].infoText3 := 'infoText3';
	ManualFnc[0].infoText4 := 'infoText4';
	ManualFnc[0].error := FALSE;
	
	ManualFnc[0].left.key.text := 'left.key.text';
	ManualFnc[0].left.status.text := 'left.status.text';
	ManualFnc[0].left.key.disable := TRUE;
	ManualFnc[0].left.status.colorChange := TRUE;
	
	ManualFnc[0].right.key.text := 'right.key.text';
	ManualFnc[0].right.status.text := 'right.status.text';
	ManualFnc[0].right.key.colorChange := TRUE;

	
	

	ManualFnc[1].headerText := 'HeaderText 2';
	ManualFnc[1].addText := '';
	ManualFnc[1].infoText1 := 'infoText1';
	ManualFnc[1].infoText2 := 'infoText2';
	ManualFnc[1].infoText3 := 'infoText3';
	ManualFnc[1].infoText4 := 'infoText4';
	ManualFnc[1].error := FALSE;
	ManualFnc[1].select := FALSE;
		
	ManualFnc[1].left.key.text := 'left.key.text';
	ManualFnc[1].left.status.text := 'left.status.text';
	ManualFnc[1].left.key.disable := FALSE;
	ManualFnc[1].left.status.colorChange := FALSE;
	
	ManualFnc[1].right.key.text := 'right.key.text';
	ManualFnc[1].right.status.text := 'right.status.text';
	ManualFnc[1].right.key.colorChange := FALSE;
	



	
	ManualFnc[2].headerText := 'HeaderText 3';
	ManualFnc[2].addText := 'addText';
	ManualFnc[2].infoText1 := 'infoText1';
	ManualFnc[2].infoText2 := 'infoText2';
	ManualFnc[2].infoText3 := 'infoText3';
	ManualFnc[2].infoText4 := 'infoText4';
	ManualFnc[2].error := TRUE;
	
	ManualFnc[2].left.key.text := 'left.key.text';
	ManualFnc[2].left.status.text := 'left.status.text';
	ManualFnc[2].left.key.disable := TRUE;
	ManualFnc[2].left.status.colorChange := TRUE;
	
	ManualFnc[2].right.key.text := 'right.key.text';
	ManualFnc[2].right.status.text := 'right.status.text';
	ManualFnc[2].right.key.colorChange := TRUE;	
	


	
	
	ManualFnc[3].headerText := 'HeaderText 4';
	ManualFnc[3].addText := '';
	ManualFnc[3].infoText1 := 'infoText1';
	ManualFnc[3].infoText2 := 'infoText2';
	ManualFnc[3].infoText3 := 'infoText3';
	ManualFnc[3].infoText4 := 'infoText4';
	ManualFnc[3].error := FALSE;
	ManualFnc[3].select := FALSE;	
	
	ManualFnc[3].left.key.text := 'left.key.text';
	ManualFnc[3].left.status.text := 'left.status.text';
	ManualFnc[3].left.key.disable := FALSE;
	ManualFnc[3].left.status.colorChange := FALSE;
	
	ManualFnc[3].right.key.text := 'right.key.text';
	ManualFnc[3].right.status.text := 'right.status.text';
	ManualFnc[3].right.key.colorChange := FALSE;

END_PROGRAM

// ---- Messages/FB_ExtSimpleEventLog.TcPOU
///****************************************************************************************
///Name:				FB_ExtSimpleEventLog
///Date:				13.10.2004
///Author:			Dirk Nordberg (BECKHOFF INDUSTRIE ELEKTRONIK)
///
///Description: Function block to control the EventLogger
///	Messages can be activated or deactivated through an array of bool.
///	The subscription of the array is equivalent to EventID from EventLogger.
///	Function block will be initialized with Init flag, then the busy flag is set true. 
///
///	Revision:	2.0
///	History:	13.10.2004	Ng	start coding
///				17.04.2005	MK	runtime optimized
///				06.09.2005 	MiB extended version (renamed to FB_ExtSimpleEventLog)
///				30.05.2017	TV  messages with format parameters
///****************************************************************************************
FUNCTION_BLOCK FB_ExtSimpleEventLog
VAR_INPUT
	/// Rising flag starts the initialization 
	Init: BOOL;
	SourceId: UINT;
	/// Alarm error class 
	Class: UINT;
	/// Activate or deaktivate confirmation 
	QuitRequired: BOOL;
	/// Adress of the array for the messages 
	adrAlarmArray: POINTER TO BOOL;
	/// ...with constant boundaries ARRAY_LBOUND to ARRAY_UBOUND for array size 
	adrQuitArray: POINTER TO BOOL;
	/// ...with constant boundaries ARRAY_LBOUND to ARRAY_UBOUND for array size 
	adrEventData: POINTER TO ST_EventData;
	/// Format String for message 
	sFormatString: STRING := '';
END_VAR
VAR_OUTPUT
	Busy: BOOL;
	Err: BOOL;
	ErrId: UDINT;
END_VAR
VAR CONSTANT
	ARRAY_LBOUND: UDINT := FIRST_MESSAGE;
	ARRAY_UBOUND: UDINT := LAST_MESSAGE;
	TCEVENTDATAFORMATSTRING: STRING(80) := ' ';
	STATE_INIT: INT := 0;
	STATE_IDLE: INT := 1;
	STATE_RESET_EVENT: INT := 2;
	STATE_QUIT_EVENT: INT := 3;
	STATE_RESET_END: INT := 4;
	STATE_WAIT: INT := 5;
END_VAR
VAR
	state: INT;
	///{flag nowatch on }
	bReady: BOOL;
	nMsgHasChanged: DINT;
	bEvtState: ARRAY[ARRAY_LBOUND..ARRAY_UBOUND] OF BOOL;
	event: ARRAY[ARRAY_LBOUND..ARRAY_UBOUND] OF ADSLOGEVENT;
	idx: UDINT;
	CfgEvent: TcEvent;
	bWait: BOOL;
	ptAlarm: POINTER TO BOOL;
	ptQuit: POINTER TO BOOL;
	RT_Init: R_TRIG;
	ptData: POINTER TO ST_EventData;
	stDummy: ST_EventData;
END_VAR

nMsgHasChanged := MEMCMP(ADR(bEvtState), adrAlarmArray, SIZEOF(bEvtState));
RT_Init(CLK:=Init);

CASE State OF
	STATE_INIT:		(* Set the parameter for TcEvent *)
		Err := FALSE;
		ErrId :=0;
		Busy := FALSE;
		CfgEvent.Prio := 0;
		CfgEvent.DataFormatStrAddress := ADR(TCEVENTDATAFORMATSTRING);
		CfgEvent.Flags := TCEVENTFLAG_LOG OR TCEVENTFLAG_SRCID;
		CfgEvent.StreamType := TCEVENTSTREAM_SIMPLE;
		CfgEvent.ProgId := 'TcEventFormatter.TcXmlFormatter';
		CfgEvent.SourceId := SourceId;
		CfgEvent.Class := Class ; 
		CfgEvent.bQuitRequired := QuitRequired;
		FOR idx := ARRAY_LBOUND TO ARRAY_UBOUND BY 1 DO
			CfgEvent.Id := idx;
			event[idx](NETID:='', PORT:=110, Event:=FALSE , EventQuit:=FALSE,
				 EventConfigData:=CfgEvent, FbCleanup:=FALSE, TMOUT:=t#1s);
		END_FOR;
		State := STATE_IDLE;

	STATE_IDLE:
		(* nothing to do *)
		IF nMsgHasChanged = 0 AND NOT RT_Init.Q THEN
			RETURN;
		END_IF

		IF adrAlarmArray <> 0 THEN
			ptAlarm := adrAlarmArray;
			ptData := adrEventData;
			IF ptData <> 0 THEN
				sFormatString := '%d%s';
				FOR idx := ARRAY_LBOUND TO ARRAY_UBOUND BY 1 DO					
					event[idx].EventConfigData.DataFormatStrAddress := ADR(sFormatString);					
					event[idx].EventConfigData.SourceId := SourceId;
					event[idx].EventDataAddress :=  ptData ; 
					event[idx].EventDataLength := SIZEOF(stDummy);
					event[idx]();
					ptData := ptData + SIZEOF(stDummy);
				END_FOR
			END_IF
			IF CfgEvent.bQuitRequired AND adrQuitArray <> 0 THEN
				ptQuit := adrQuitArray;
				FOR idx := ARRAY_LBOUND TO ARRAY_UBOUND BY 1 DO
					event[idx](Event:=ptAlarm^, EventQuit:=ptQuit^);
					ptAlarm := ptAlarm + 1;
					ptQuit := ptQuit + 1;
				END_FOR;
			ELSE
				bReady := TRUE;
				FOR idx := ARRAY_LBOUND TO ARRAY_UBOUND BY 1 DO
					event[idx](Event:=ptAlarm^);
					ptAlarm := ptAlarm + 1;
					IF (NOT(event[idx].Event = TRUE			(* event is set *)
							AND event[idx].Quit = FALSE
							AND event[idx].EventState = TCEVENTSTATE_SIGNALED)
						AND NOT(event[idx].Event = FALSE		(* event is reset *)
							AND event[idx].Quit = TRUE
							AND event[idx].EventState = TCEVENTSTATE_INVALID)) THEN
						bReady := FALSE;
					END_IF
				END_FOR;

				(* copy the status *)
				IF bReady THEN
					MEMCPY(ADR(bEvtState), adrAlarmArray, SIZEOF(bEvtState));
				END_IF

			END_IF
		END_IF

		IF RT_Init.Q THEN
			Busy := TRUE;
			State := STATE_RESET_EVENT;
		END_IF

	STATE_RESET_EVENT:(*---------------------------------- clear messages ----------------------------------------*)
		FOR idx := ARRAY_LBOUND TO ARRAY_UBOUND BY 1 DO
			IF event[idx].EventState = TCEVENTSTATE_SIGNALED THEN
				event[idx](Event:=FALSE, EventQuit:= FALSE, FbCleanup:= FALSE, TMOUT:= t#1s);
				IF event[idx].Err THEN
					Err := TRUE;
					ErrId := event[idx].ErrId;
					IF event[idx].ErrId = 1282 THEN	(* Message Router: mailbox full *)
						event[idx](Event:=FALSE, EventQuit:= FALSE, FbCleanup:= FALSE);
						RETURN;
					END_IF
				END_IF
			END_IF;
		END_FOR;
		State := STATE_QUIT_EVENT;

	STATE_QUIT_EVENT:(*---------------------------------- quit messages ----------------------------------------*)
		FOR idx := ARRAY_LBOUND TO ARRAY_UBOUND BY 1 DO
			IF event[idx].EventState = TCEVENTSTATE_SIGNALED THEN
				event[idx](Event:=FALSE, EventQuit:= TRUE, FbCleanup:= FALSE, TMOUT:= t#1s);
				IF event[idx].Err THEN
					Err := TRUE;
					ErrId := event[idx].ErrId;
					IF event[idx].ErrId = 1282 THEN	(* Message Router: mailbox full *)
						event[idx](Event:=FALSE, EventQuit:= FALSE, FbCleanup:= FALSE);
						RETURN;
					END_IF
				END_IF
			END_IF;
		END_FOR;
		State := STATE_RESET_END;

	STATE_RESET_END:
		bWait := FALSE;
		FOR idx := ARRAY_LBOUND TO ARRAY_UBOUND BY 1 DO
			event[idx](Event:=FALSE, EventQuit:= FALSE, FbCleanup:= FALSE);
			IF event[idx].EventState = TCEVENTSTATE_SIGNALED THEN
				bWait := TRUE;
			END_IF
		END_FOR;
		IF NOT bWait THEN
			State := STATE_INIT;
		END_IF

END_CASE

END_FUNCTION_BLOCK

// ---- Samples/PRG_FastMFunctions.TcPOU
PROGRAM PRG_FastMFunctions
VAR
	anMFunctionNo						: ARRAY[0..MAX_FAST_M_FUNC_ITEM_IDX] OF UINT;	
	fbFastMFunctionProvider				: HLI3_FastMFunctionProvider;
	fbFastMFunctionHandler				: HLI3_FastMFunctionHandler;	
	abyOutput					AT %Q*	: ARRAY[0..MAX_FAST_M_FUNC_OUTPUT_IDX] OF BYTE;  	
END_VAR

(****************************************************************************************)
(* POU:		PRG_FastMFunctions                    										*)
(* Type:	PRG																			*)
(* Author: 	RCH		                                             						*)
(* Date: 	14/10/29																	*)
(* Rev.: 	1.0                                               							*)
(* ------------------------------------------------------------------------------------ *)
(* Desc.:	PLC program to demonstrate usage of MOS_TS M functions using the FB´s		*)
(*			HLI3_FastMFunctionProvider and HLI3_FastMFunctionHandler.					*)
(*			In order to achieve a determenistic output behavior this program has to be 	*)
(*			called by a task running synchronously to the CNC GEO task. Therefore that	*)
(*			task´s priority  has to be adjusted in a way that it gets called by the 	*)
(* 			realtime system	right after the CNC GEO task.								*)
(*																						*)
(*			THIS IMPLEMENTATION REQUIRES A 1MS CNC GEO AND 1MS FAST PLC TASK CYCLE!!!	*)
(* ------------------------------------------------------------------------------------ *)
(* Rev.:	<Enter revision number here>												*)
(* Date:	<Enter revision data here>				                                   	*)
(* Author:	<Enter author´s shortcut here>											 	*)
(* Desc.:	<Enter description here>													*)
(****************************************************************************************)


(****************************************************************************************)
(*	  						Configure M function no´s to provide						*)
(****************************************************************************************)
(* Add up to MAX_FAST_M_FUNC_ITEM_IDX m function numbers that should be handled by 		*)
(* fbFastMFunctionProvider.																*)
anMFunctionNo[0]	:= 25;
anMFunctionNo[1]	:= 26;

fbFastMFunctionProvider
	(nHliChanIdx	:= 0, 
	 anMFunctionNo	:= anMFunctionNo
	);
	
(****************************************************************************************)
(*	  						 	Handle Laser ON/OFF (M25/M26)							*)
(****************************************************************************************)
(* M function numbers for switching ON and OFF have to be contained in the 				*)
(* 'anMFunctionNo' array of the HLI3_FastMFunctionProvider instance which provides the	*)
(* 'stData' structure to this FB.														*)
(* The delay times nDelayOn and nDelayOff can be used to adopt to external hardware		*)
(* delays!																				*)
fbFastMFunctionHandler
	(bForceOff		:= FALSE, 
	 bReset			:= FALSE, 
	 nFunctionNoOn	:= 25, 
	 nDelayOn		:= 0,			
	 nFunctionNoOff	:= 26, 
	 nDelayOff		:= 0,
	 stData			:= fbFastMFunctionProvider.stData,
	 abyOutput		=> abyOutput
	);

END_PROGRAM
